(* IEC 61131-3 sources: Word/plc-course/13-sequential-control/labs/solutions, 3 files *)

(* ---- 13-1-pedestrian-crossing.st ---- *)
(* Lab 13-1: Pedestrian crossing as a CASE state machine.
   Module 13 (Sequential control). REFERENCE SOLUTION - try the lab yourself first.

   The crossing rests on vehicle green. A pedestrian request is remembered,
   and it is served only after the vehicles have had their minimum green.
   The program has four parts, always in this order:
     1. step bookkeeping: an entry flag and ONE step timer, reset on every
        change of state
     2. the CASE: one branch per state, containing only its transitions
     3. things that are remembered between states (the request latch, the
        flasher)
     4. outputs derived from the state: exactly one assignment per output *)

TYPE
  E_Crossing : (Startup, RedAmber, Green, Amber, AllRed, Walk, PedClear);
END_TYPE

PROGRAM PedCrossing
  VAR (* I/O *)
    PedPB    AT %IX0.0 : BOOL;  (* pedestrian request push-button, NO *)
    CarRed   AT %QX0.0 : BOOL;  (* vehicle signal, red *)
    CarAmber AT %QX0.1 : BOOL;  (* vehicle signal, amber *)
    CarGreen AT %QX0.2 : BOOL;  (* vehicle signal, green *)
    PedRed   AT %QX0.3 : BOOL;  (* pedestrian signal, red figure: do not cross *)
    PedGreen AT %QX0.4 : BOOL;  (* pedestrian signal, green figure: cross *)
    WaitLamp AT %QX0.5 : BOOL;  (* WAIT lamp on the push-button box *)
  END_VAR
  VAR (* settings *)
    StartupTime  : TIME := T#3s;   (* all red after power-up *)
    RedAmberTime : TIME := T#2s;   (* red + amber before green *)
    MinGreen     : TIME := T#10s;  (* minimum vehicle green *)
    AmberTime    : TIME := T#3s;   (* amber after green *)
    AllRedTime   : TIME := T#2s;   (* all red before the walk phase *)
    WalkTime     : TIME := T#6s;   (* steady green figure *)
    PedClearTime : TIME := T#4s;   (* flashing green figure *)
  END_VAR
  VAR (* internal *)
    State      : E_Crossing := Startup;
    PrevState  : E_Crossing := Startup;
    FirstScan  : BOOL := TRUE;
    StepEntry  : BOOL;           (* TRUE on the first scan in a state *)
    StepTimer  : TON;            (* time spent in the current state *)
    Request    : BOOL;           (* latched pedestrian request *)
    FlashTimer : TON;            (* 500 ms flasher for the clearance phase *)
    FlashOn    : BOOL;
  END_VAR

  (* 1. Step bookkeeping. StepEntry is TRUE for exactly one scan after every
        change of state (and on the very first scan). Calling the step timer
        with IN := NOT StepEntry resets it for that scan, so StepTimer.ET
        always means "time in the current state". *)
  StepEntry := (State <> PrevState) OR FirstScan;
  FirstScan := FALSE;
  PrevState := State;
  StepTimer(IN := NOT StepEntry, PT := T#24h);

  (* 2. Transitions. Only the branch of the current state runs, so the
        crossing can move at most one state per scan. *)
  CASE State OF
    Startup:
      IF StepTimer.ET >= StartupTime THEN
        State := RedAmber;
      END_IF;

    RedAmber:
      IF StepTimer.ET >= RedAmberTime THEN
        State := Green;
      END_IF;

    Green:
      (* rest here until someone asks, but always give the minimum green *)
      IF Request AND (StepTimer.ET >= MinGreen) THEN
        State := Amber;
      END_IF;

    Amber:
      IF StepTimer.ET >= AmberTime THEN
        State := AllRed;
      END_IF;

    AllRed:
      IF StepTimer.ET >= AllRedTime THEN
        State := Walk;
      END_IF;

    Walk:
      IF StepTimer.ET >= WalkTime THEN
        State := PedClear;
      END_IF;

    PedClear:
      IF StepTimer.ET >= PedClearTime THEN
        State := RedAmber;
      END_IF;
  ELSE
    (* An impossible value: restart through the all-red start-up phase. *)
    State := Startup;
  END_CASE;

  (* 3a. Request latch. A press is remembered in every state except Walk,
         where the pedestrians already have their green. The latch is
         cleared in the same scan as the walk phase starts, so the WAIT lamp
         goes out exactly when the green figure lights. *)
  Request := (Request OR PedPB) AND (State <> Walk);

  (* 3b. Flasher for the clearance phase: toggles every 500 ms and starts
         with the green figure OFF, so pedestrians see the change at once. *)
  FlashTimer(IN := (State = PedClear) AND NOT FlashTimer.Q, PT := T#500ms);
  IF State <> PedClear THEN
    FlashOn := FALSE;
  ELSIF FlashTimer.Q THEN
    FlashOn := NOT FlashOn;
  END_IF;

  (* 4. Outputs, derived from the state. Reading down a column of the lab's
        state/output table gives each of these lines. *)
  CarRed   := (State = Startup) OR (State = RedAmber)
           OR (State = AllRed) OR (State = Walk)
           OR (State = PedClear);
  CarAmber := (State = RedAmber) OR (State = Amber);
  CarGreen := State = Green;
  PedGreen := (State = Walk) OR ((State = PedClear) AND FlashOn);
  PedRed   := (State <> Walk) AND (State <> PedClear);
  WaitLamp := Request;
END_PROGRAM

CONFIGURATION Config0
  RESOURCE Res0 ON PLC
    TASK MainTask(INTERVAL := T#10ms, PRIORITY := 0);
    PROGRAM Inst0 WITH MainTask : PedCrossing;
  END_RESOURCE
END_CONFIGURATION

(* ---- 13-2-batch-tank.st ---- *)
(* Lab 13-2: Batch tank sequence with watchdogs, Hold/Resume and Abort.
   Module 13 (Sequential control). REFERENCE SOLUTION - try the lab yourself first.

   Fill -> Mix -> Heat -> Drain, as a CASE state machine. Every step that
   waits for the plant has a watchdog that leads to a fault state. Hold
   parks the batch safely and Resume returns to the step it came from;
   Abort ends the batch from any running or held state.

   Order of the program:
     1. operator commands (rising edges)
     2. step bookkeeping: entry flag and step timer
     3. entry actions
     4. transitions: Abort, then Hold, then the step's own transitions
     5. outputs derived from the state, plus interlocks that apply in
        every state *)

TYPE
  E_Batch : (Idle, Filling, Mixing, Heating, Draining, Complete, Held, Faulted);
END_TYPE

PROGRAM BatchTank
  VAR (* I/O *)
    StartPB      AT %IX0.0 : BOOL;  (* start a batch, NO *)
    HoldPB       AT %IX0.1 : BOOL;  (* hold the batch, NO *)
    ResumePB     AT %IX0.2 : BOOL;  (* resume a held batch, NO *)
    AbortPB      AT %IX0.3 : BOOL;  (* abort the batch, NO *)
    ResetPB      AT %IX0.4 : BOOL;  (* fault reset, NO *)
    LevelHighLS  AT %IX0.5 : BOOL;  (* high-level switch: TRUE when the tank is full *)
    LevelLowLS   AT %IX0.6 : BOOL;  (* low-level switch: TRUE while liquid covers it (and the heater) *)
    InletValve   AT %QX0.0 : BOOL;  (* fill valve *)
    Agitator     AT %QX0.1 : BOOL;  (* mixer motor *)
    Heater       AT %QX0.2 : BOOL;  (* immersion heater contactor *)
    OutletValve  AT %QX0.3 : BOOL;  (* drain valve *)
    RunLamp      AT %QX0.4 : BOOL;  (* batch running *)
    HeldLamp     AT %QX0.5 : BOOL;  (* batch held *)
    FaultLamp    AT %QX0.6 : BOOL;  (* sequence fault *)
    CompleteLamp AT %QX0.7 : BOOL;  (* batch complete *)
  END_VAR
  VAR (* process value, written by the analog-input layer (Module 14) *)
    TankTemp : REAL;                (* tank temperature, degC *)
  END_VAR
  VAR (* settings *)
    TempSP       : REAL := 60.0;    (* heat until TankTemp >= TempSP *)
    MixTime      : TIME := T#10s;   (* total mixing time *)
    FillTimeout  : TIME := T#30s;   (* watchdog: filling *)
    HeatTimeout  : TIME := T#60s;   (* watchdog: heating *)
    DrainTimeout : TIME := T#30s;   (* watchdog: draining *)
  END_VAR
  VAR (* status for the HMI *)
    FaultCode  : INT;               (* 0 none, 1 fill, 2 heat, 3 drain timeout *)
    BatchCount : INT;               (* completed batches *)
  END_VAR
  VAR (* internal *)
    State     : E_Batch := E_Batch#Idle;
    PrevState : E_Batch := E_Batch#Idle;
    HeldFrom  : E_Batch := E_Batch#Idle;  (* the step to resume *)
    FirstScan : BOOL := TRUE;
    StepEntry : BOOL;               (* TRUE on the first scan in a state *)
    StepTimer : TON;                (* time in the current state *)
    MixDone   : TIME;               (* mixing completed before a hold *)
    Running   : BOOL;               (* in one of the four process steps *)
    (* One instance per line: OpenPLC's compiler can crash on a list of
       FB instances in one declaration (see Appendix E). *)
    StartEdge : R_TRIG;
    HoldEdge : R_TRIG;
    ResumeEdge : R_TRIG;
    AbortEdge : R_TRIG;
    ResetEdge : R_TRIG;
    StartCmd, HoldCmd, ResumeCmd, AbortCmd, ResetCmd : BOOL;
  END_VAR

  (* 1. Commands act once per press. A button that is already held when the
        PLC starts is not treated as a press. *)
  StartEdge(CLK := StartPB);
  HoldEdge(CLK := HoldPB);
  ResumeEdge(CLK := ResumePB);
  AbortEdge(CLK := AbortPB);
  ResetEdge(CLK := ResetPB);
  StartCmd  := StartEdge.Q AND NOT FirstScan;
  HoldCmd   := HoldEdge.Q AND NOT FirstScan;
  ResumeCmd := ResumeEdge.Q AND NOT FirstScan;
  AbortCmd  := AbortEdge.Q AND NOT FirstScan;
  ResetCmd  := ResetEdge.Q AND NOT FirstScan;

  (* 2. Step bookkeeping: StepEntry is TRUE for one scan after each change,
        and the step timer restarts from zero on every entry. *)
  StepEntry := (State <> PrevState) OR FirstScan;
  FirstScan := FALSE;
  PrevState := State;
  StepTimer(IN := NOT StepEntry, PT := T#24h);

  (* 3. Entry actions: done once, on the first scan in a state. They come
        BEFORE the transitions, because StepEntry belongs to the state the
        scan started in. *)
  IF StepEntry AND (State = E_Batch#Complete) THEN
    BatchCount := BatchCount + 1;
  END_IF;

  Running := (State = E_Batch#Filling) OR (State = E_Batch#Mixing)
          OR (State = E_Batch#Heating) OR (State = E_Batch#Draining);

  (* 4. Transitions. Abort beats Hold, and both beat the step's own
        transitions, so they are tested first. *)
  IF AbortCmd AND (Running OR (State = E_Batch#Held)) THEN
    State := E_Batch#Idle;

  ELSIF HoldCmd AND Running THEN
    IF State = E_Batch#Mixing THEN
      (* bank the mixing done so far: it still counts after Resume *)
      MixDone := ADD_TIME(MixDone, StepTimer.ET);
    END_IF;
    HeldFrom := State;
    State := E_Batch#Held;

  ELSE
    CASE State OF
      E_Batch#Idle, E_Batch#Complete:
        IF StartCmd THEN
          MixDone := T#0s;
          State := E_Batch#Filling;
        END_IF;

      E_Batch#Filling:
        IF LevelHighLS THEN
          State := E_Batch#Mixing;
        ELSIF StepTimer.ET >= FillTimeout THEN
          FaultCode := 1;
          State := E_Batch#Faulted;
        END_IF;

      E_Batch#Mixing:
        IF ADD_TIME(MixDone, StepTimer.ET) >= MixTime THEN
          State := E_Batch#Heating;
        END_IF;

      E_Batch#Heating:
        IF TankTemp >= TempSP THEN
          State := E_Batch#Draining;
        ELSIF StepTimer.ET >= HeatTimeout THEN
          FaultCode := 2;
          State := E_Batch#Faulted;
        END_IF;

      E_Batch#Draining:
        IF NOT LevelLowLS THEN
          State := E_Batch#Complete;
        ELSIF StepTimer.ET >= DrainTimeout THEN
          FaultCode := 3;
          State := E_Batch#Faulted;
        END_IF;

      E_Batch#Held:
        IF ResumeCmd THEN
          State := HeldFrom;        (* its step timer and watchdog restart *)
        END_IF;

      E_Batch#Faulted:
        IF ResetCmd THEN
          FaultCode := 0;
          State := E_Batch#Idle;    (* the operator decides what happens next *)
        END_IF;
    ELSE
      FaultCode := 99;              (* impossible state value: stop safely *)
      State := E_Batch#Faulted;
    END_CASE;
  END_IF;

  (* 5. Outputs from the state (recomputed after the transitions, so an
        output changes in the same scan as its state). The interlocks are
        written here, separately from the sequence, so they hold whatever
        state the sequence is in. *)
  Running := (State = E_Batch#Filling) OR (State = E_Batch#Mixing)
          OR (State = E_Batch#Heating) OR (State = E_Batch#Draining);

  InletValve  := (State = E_Batch#Filling) AND NOT LevelHighLS;  (* never overfill *)
  Agitator    := (State = E_Batch#Mixing) OR (State = E_Batch#Heating);
  Heater      := (State = E_Batch#Heating) AND LevelLowLS;       (* elements covered *)
  OutletValve := State = E_Batch#Draining;

  RunLamp      := Running;
  HeldLamp     := State = E_Batch#Held;
  FaultLamp    := State = E_Batch#Faulted;
  CompleteLamp := State = E_Batch#Complete;
END_PROGRAM

CONFIGURATION Config0
  RESOURCE Res0 ON PLC
    TASK MainTask(INTERVAL := T#10ms, PRIORITY := 0);
    PROGRAM Inst0 WITH MainTask : BatchTank;
  END_RESOURCE
END_CONFIGURATION

(* ---- 13-3-drill-sfc.st ---- *)
(* Lab 13-3: Drilling station in textual SFC, with action qualifiers.
   Module 13 (Sequential control). REFERENCE SOLUTION - try the lab yourself first.

   The whole program body is a Sequential Function Chart written in the
   textual form of IEC 61131-3 (the form MATIEC compiles, and the form the
   OpenPLC Editor generates from a graphical chart).

        Idle          ReadyLamp(N)
          + StartPB AND PartPE AND DrillUpLS
        Clamp         ClampValve(S)
          + ClampedLS
        Drill         Spindle(S), FeedDown(D, SpinUpTime)
          + DrillDownLS                 + NOT DrillDownLS AND Drill.T >= FeedTimeout
        Dwell         CountHole(P)      FeedFault   FaultLamp(N), Spindle(R)
          + Dwell.T >= DwellTime          + ResetPB  (jump to Retract)
        Retract       FeedUp(N), BlowAir(L, BlowTime)
          + DrillUpLS
        Unclamp       Spindle(R), ClampValve(R)
          + NOT ClampedLS
        Unload        (waits for the part to be taken out)
          + NOT PartPE  (jump back to Idle)

   Why these qualifiers:
     S/R  the clamp and the spindle stay on across several steps, so they
          are set in one step and reset in a later one;
     D    the feed starts only after the spindle has run up to speed;
     L    the chip blow-off lasts at most BlowTime, and stops earlier if the
          drill reaches the top first;
     P    the hole counter is incremented once, when the Dwell step starts;
     N    everything else is on exactly while its step is active.
   The two transitions out of Drill are written to be mutually exclusive:
   MATIEC fires every enabled transition whose condition is TRUE. *)

PROGRAM DrillCycle
  VAR (* I/O *)
    StartPB     AT %IX0.0 : BOOL;  (* cycle start push-button, NO *)
    PartPE      AT %IX0.1 : BOOL;  (* part present in the fixture *)
    ClampedLS   AT %IX0.2 : BOOL;  (* clamp closed *)
    DrillUpLS   AT %IX0.3 : BOOL;  (* drill head at the top (home) *)
    DrillDownLS AT %IX0.4 : BOOL;  (* drill at full depth *)
    ResetPB     AT %IX0.5 : BOOL;  (* fault reset push-button, NO *)
    ClampValve  AT %QX0.0 : BOOL;  (* clamp solenoid valve: TRUE = clamp *)
    Spindle     AT %QX0.1 : BOOL;  (* spindle motor contactor *)
    FeedDown    AT %QX0.2 : BOOL;  (* feed valve, down *)
    FeedUp      AT %QX0.3 : BOOL;  (* feed valve, up (neither = hold position) *)
    BlowAir     AT %QX0.4 : BOOL;  (* chip blow-off air valve *)
    ReadyLamp   AT %QX0.5 : BOOL;  (* ready for a new part *)
    FaultLamp   AT %QX0.6 : BOOL;  (* feed fault *)
  END_VAR
  VAR (* settings and counters *)
    SpinUpTime  : TIME := T#500ms; (* spindle run-up before the feed starts *)
    DwellTime   : TIME := T#1s;    (* dwell at full depth *)
    BlowTime    : TIME := T#1s;    (* longest blow-off during the retract *)
    FeedTimeout : TIME := T#5s;    (* longest time allowed to reach depth *)
    HoleCount   : INT;             (* holes drilled to full depth *)
  END_VAR

  INITIAL_STEP Idle:
    ReadyLamp(N);
  END_STEP

  TRANSITION FROM Idle TO Clamp
    := StartPB AND PartPE AND DrillUpLS;
  END_TRANSITION

  STEP Clamp:
    ClampValve(S);
  END_STEP

  TRANSITION FROM Clamp TO Drill
    := ClampedLS;
  END_TRANSITION

  STEP Drill:
    Spindle(S);
    FeedDown(D, SpinUpTime);
  END_STEP

  (* Alternative branch: depth reached, or the feed watchdog. *)
  TRANSITION FROM Drill TO Dwell
    := DrillDownLS;
  END_TRANSITION

  TRANSITION FROM Drill TO FeedFault
    := NOT DrillDownLS AND (Drill.T >= FeedTimeout);
  END_TRANSITION

  STEP Dwell:
    CountHole(P);
  END_STEP

  TRANSITION FROM Dwell TO Retract
    := Dwell.T >= DwellTime;
  END_TRANSITION

  STEP Retract:
    FeedUp(N);
    BlowAir(L, BlowTime);
  END_STEP

  TRANSITION FROM Retract TO Unclamp
    := DrillUpLS;
  END_TRANSITION

  STEP Unclamp:
    Spindle(R);
    ClampValve(R);
  END_STEP

  TRANSITION FROM Unclamp TO Unload
    := NOT ClampedLS;
  END_TRANSITION

  STEP Unload:
  END_STEP

  TRANSITION FROM Unload TO Idle
    := NOT PartPE;
  END_TRANSITION

  (* Fault branch: stop the spindle and hold the feed where it is, keep the
     part clamped, and retract only when the operator resets. *)
  STEP FeedFault:
    FaultLamp(N);
    Spindle(R);
  END_STEP

  TRANSITION FROM FeedFault TO Retract
    := ResetPB;
  END_TRANSITION

  ACTION CountHole:
    HoleCount := HoleCount + 1;
  END_ACTION
END_PROGRAM

CONFIGURATION Config0
  RESOURCE Res0 ON PLC
    TASK MainTask(INTERVAL := T#10ms, PRIORITY := 0);
    PROGRAM Inst0 WITH MainTask : DrillCycle;
  END_RESOURCE
END_CONFIGURATION
